SUBAPPLICATION Uebung_071b (* WBSD auf UT ausgeben, Q1 Schalten wenn Speed >0 *)
  (* Standard: 61499-2; Description: Copyright (c) 2023 Meisterschulen am Ostbahnhof This program and the accompanying materials are made available under the terms of the Eclipse Public License 2.0 which is available at https://www.eclipse.org/legal/epl-2.0/ SPDX-License-Identifier: EPL-2.0 *)
  (* Version 1.0, 2023-10-23, Franz Höpfinger, Meisterschulen am Ostbahnhof *)
  PACKAGE Uebungen;
  IMPORT Uebungen::const::UT::DefaultPool_TECU::NumberVariable_Wheel_based_machine_distance;
  IMPORT Uebungen::const::UT::DefaultPool_TECU::NumberVariable_Wheel_based_machine_speed;
  IMPORT logiBUS::io::DQ::logiBUS_DO::Output_Q1;
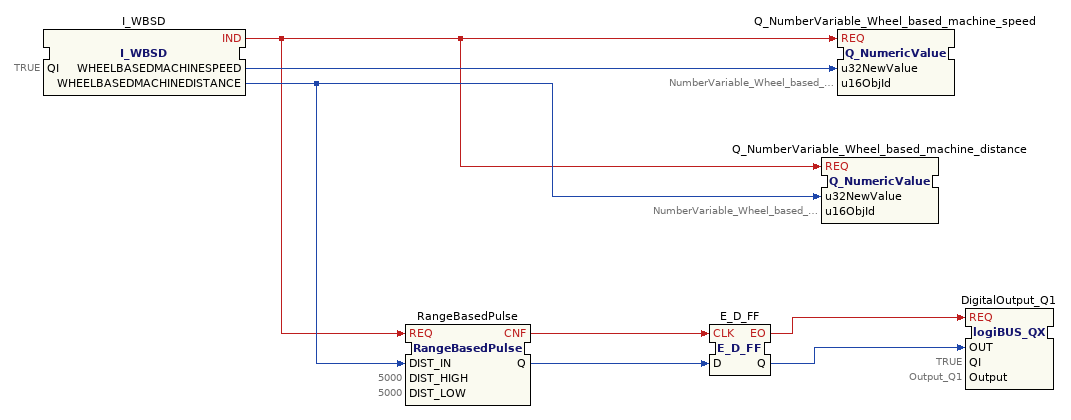
  FBS
    I_WBSD : isobus::tecu::I_WBSD(QI := TRUE);
    Q_NumberVariable_Wheel_based_machine_speed : isobus::UT::Q::Q_NumericValue(u16ObjId := NumberVariable_Wheel_based_machine_speed);
    DigitalOutput_Q1 : logiBUS::io::DQ::logiBUS_QX(QI := TRUE, Output := Output_Q1);
    RangeBasedPulse : eclipse4diac::signalprocessing::distance::RangeBasedPulse(DIST_HIGH := 5000, DIST_LOW := 5000);
    E_D_FF : iec61499::events::E_D_FF;
    Q_NumberVariable_Wheel_based_machine_distance : isobus::UT::Q::Q_NumericValue(u16ObjId := NumberVariable_Wheel_based_machine_distance);
  END_FBS
  EVENT_CONNECTIONS
    I_WBSD.IND TO Q_NumberVariable_Wheel_based_machine_speed.REQ;
    E_D_FF.EO TO DigitalOutput_Q1.REQ;
    I_WBSD.IND TO Q_NumberVariable_Wheel_based_machine_distance.REQ;
    I_WBSD.IND TO RangeBasedPulse.REQ;
    RangeBasedPulse.CNF TO E_D_FF.CLK;
  END_CONNECTIONS
  DATA_CONNECTIONS
    I_WBSD.WHEELBASEDMACHINESPEED TO Q_NumberVariable_Wheel_based_machine_speed.u32NewValue;
    E_D_FF.Q TO DigitalOutput_Q1.OUT;
    I_WBSD.WHEELBASEDMACHINEDISTANCE TO Q_NumberVariable_Wheel_based_machine_distance.u32NewValue;
    I_WBSD.WHEELBASEDMACHINEDISTANCE TO RangeBasedPulse.DIST_IN;
    RangeBasedPulse.Q TO E_D_FF.D;
  END_CONNECTIONS
END_SUBAPPLICATION
